RESOURCE_TYPE test2
  (* Standard: 61499-2 *)
  (* Version 0.1, 2016-00-15, Hammond, HAMMONDSDESKTOP *)
  VAR_INPUT
    ac1_default_var : ARRAY [0..3] OF INT := [0, 1, 2, 3];
    ac2_default_var : ARRAY [0..3] OF INT := [3, 2, 1, 0];
  END_VAR
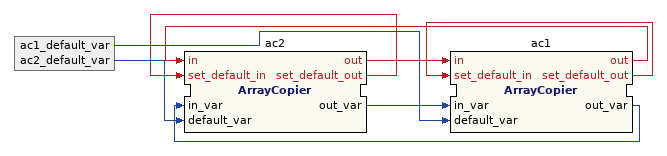
  FBS
    ac1 : ArrayCopier;
    ac2 : ArrayCopier;
  END_FBS
  EVENT_CONNECTIONS
    ac1.out TO ac2.in;
    ac1.set_default_out TO ac1.set_default_in;
    ac2.out TO ac1.in;
    ac2.set_default_out TO ac2.set_default_in;
  END_CONNECTIONS
  DATA_CONNECTIONS
    ac1_default_var TO ac1.default_var;
    ac2_default_var TO ac2.default_var;
    ac1.out_var TO ac2.in_var;
    ac2.out_var TO ac1.in_var;
  END_CONNECTIONS
END_RESOURCE_TYPE
